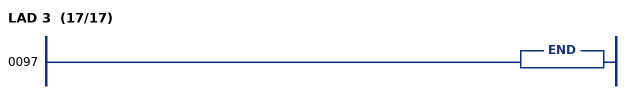
% Rung: 97 %
SOR END EOR

LADDER 4
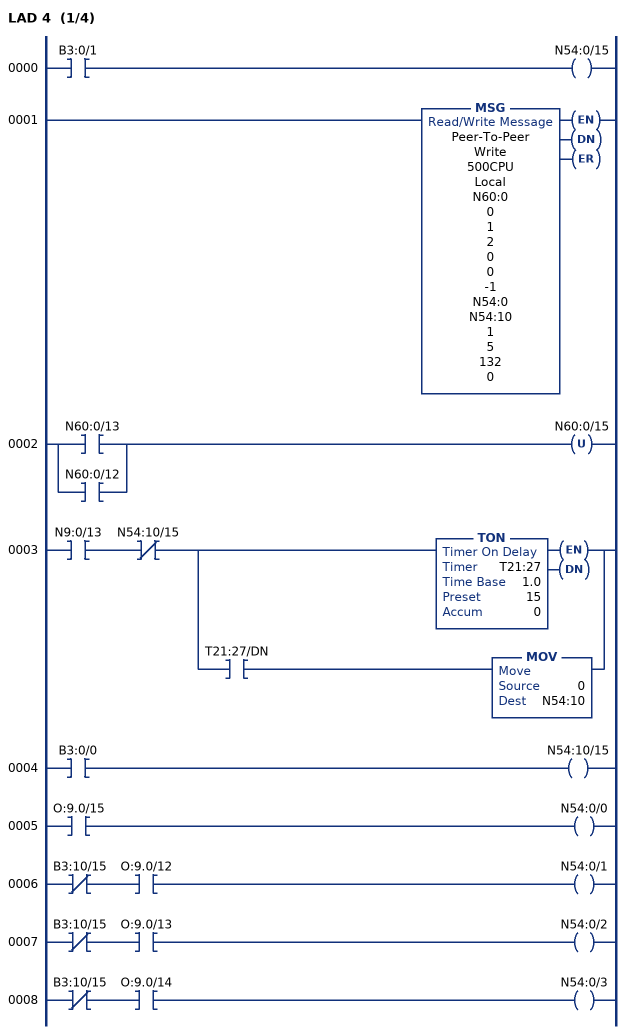
% Rung: 0 %
SOR XIC B3:0/1 OTE N54:0/15 EOR
% Rung: 1 %
SOR MSG Peer-To-Peer Write 500CPU Local N60:0 0 1 2 0 0 -1 N54:0 N54:10 1 5 132 0 EOR
%   MSG set-up: 500CPU Write | 5 | 1 | N54:10 | N54:0 | 0 | 2 | 2 | CLIENT | 0 | 0 %
% Rung: 2 %
SOR BST XIC N60:0/13 NXB XIC N60:0/12 BND OTU N60:0/15 EOR
% Rung: 3 %
SOR XIC N9:0/13 XIO N54:10/15 BST TON T21:27 1.0 15 0 NXB XIC T21:27/DN MOV 0 N54:10 BND EOR
% Rung: 4 %
SOR XIC B3:0/0 OTE N54:10/15 EOR
% Rung: 5 %
SOR XIC O:9.0/15 OTE N54:0/0 EOR
% Rung: 6 %
SOR XIO B3:10/15 XIC O:9.0/12 OTE N54:0/1 EOR
% Rung: 7 %
SOR XIO B3:10/15 XIC O:9.0/13 OTE N54:0/2 EOR
% Rung: 8 %
SOR XIO B3:10/15 XIC O:9.0/14 OTE N54:0/3 EOR

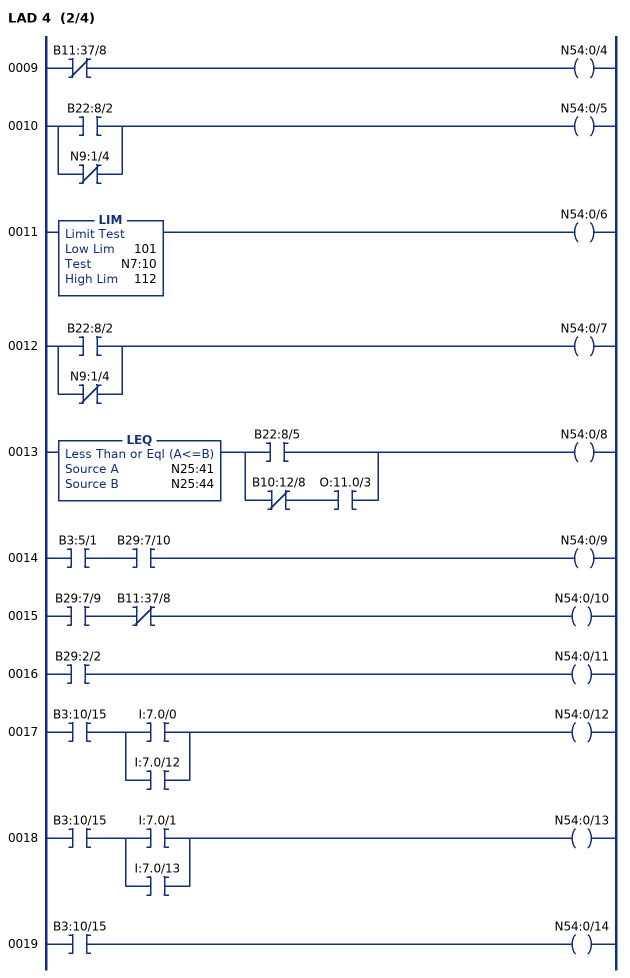
% Rung: 9 %
SOR XIO B11:37/8 OTE N54:0/4 EOR
% Rung: 10 %
SOR BST XIC B22:8/2 NXB XIO N9:1/4 BND OTE N54:0/5 EOR
% Rung: 11 %
SOR LIM 101 N7:10 112 OTE N54:0/6 EOR
% Rung: 12 %
SOR BST XIC B22:8/2 NXB XIO N9:1/4 BND OTE N54:0/7 EOR
% Rung: 13 %
SOR LEQ N25:41 N25:44 BST XIC B22:8/5 NXB XIO B10:12/8 XIC O:11.0/3 BND OTE N54:0/8 EOR
% Rung: 14 %
SOR XIC B3:5/1 XIC B29:7/10 OTE N54:0/9 EOR
% Rung: 15 %
SOR XIC B29:7/9 XIO B11:37/8 OTE N54:0/10 EOR
% Rung: 16 %
SOR XIC B29:2/2 OTE N54:0/11 EOR
% Rung: 17 %
SOR XIC B3:10/15 BST XIC I:7.0/0 NXB XIC I:7.0/12 BND OTE N54:0/12 EOR
% Rung: 18 %
SOR XIC B3:10/15 BST XIC I:7.0/1 NXB XIC I:7.0/13 BND OTE N54:0/13 EOR
% Rung: 19 %
SOR XIC B3:10/15 OTE N54:0/14 EOR

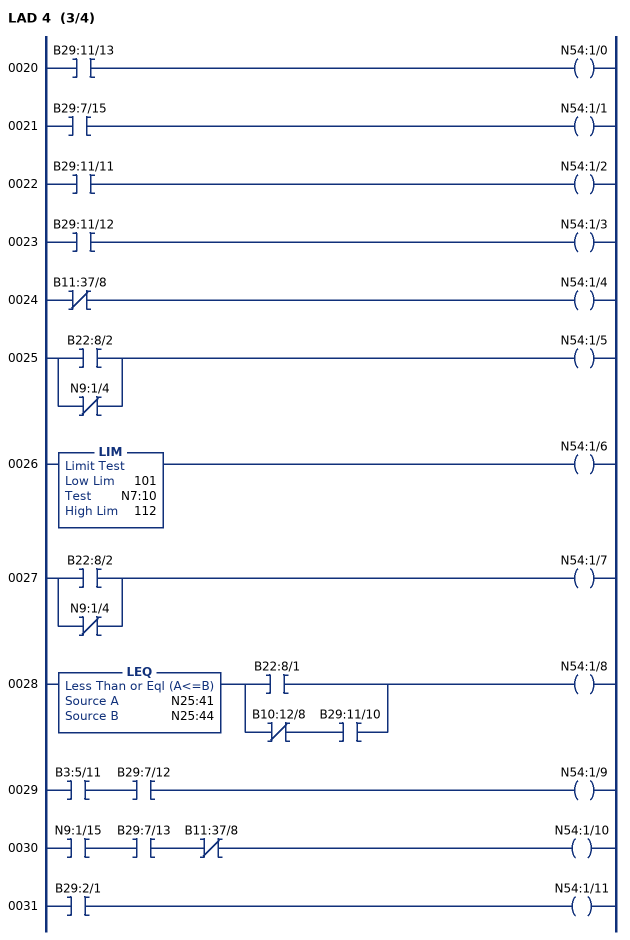
% Rung: 20 %
SOR XIC B29:11/13 OTE N54:1/0 EOR
% Rung: 21 %
SOR XIC B29:7/15 OTE N54:1/1 EOR
% Rung: 22 %
SOR XIC B29:11/11 OTE N54:1/2 EOR
% Rung: 23 %
SOR XIC B29:11/12 OTE N54:1/3 EOR
% Rung: 24 %
SOR XIO B11:37/8 OTE N54:1/4 EOR
% Rung: 25 %
SOR BST XIC B22:8/2 NXB XIO N9:1/4 BND OTE N54:1/5 EOR
% Rung: 26 %
SOR LIM 101 N7:10 112 OTE N54:1/6 EOR
% Rung: 27 %
SOR BST XIC B22:8/2 NXB XIO N9:1/4 BND OTE N54:1/7 EOR
% Rung: 28 %
SOR LEQ N25:41 N25:44 BST XIC B22:8/1 NXB XIO B10:12/8 XIC B29:11/10 BND OTE N54:1/8 EOR
% Rung: 29 %
SOR XIC B3:5/11 XIC B29:7/12 OTE N54:1/9 EOR
% Rung: 30 %
SOR XIC N9:1/15 XIC B29:7/13 XIO B11:37/8 OTE N54:1/10 EOR
% Rung: 31 %
SOR XIC B29:2/1 OTE N54:1/11 EOR

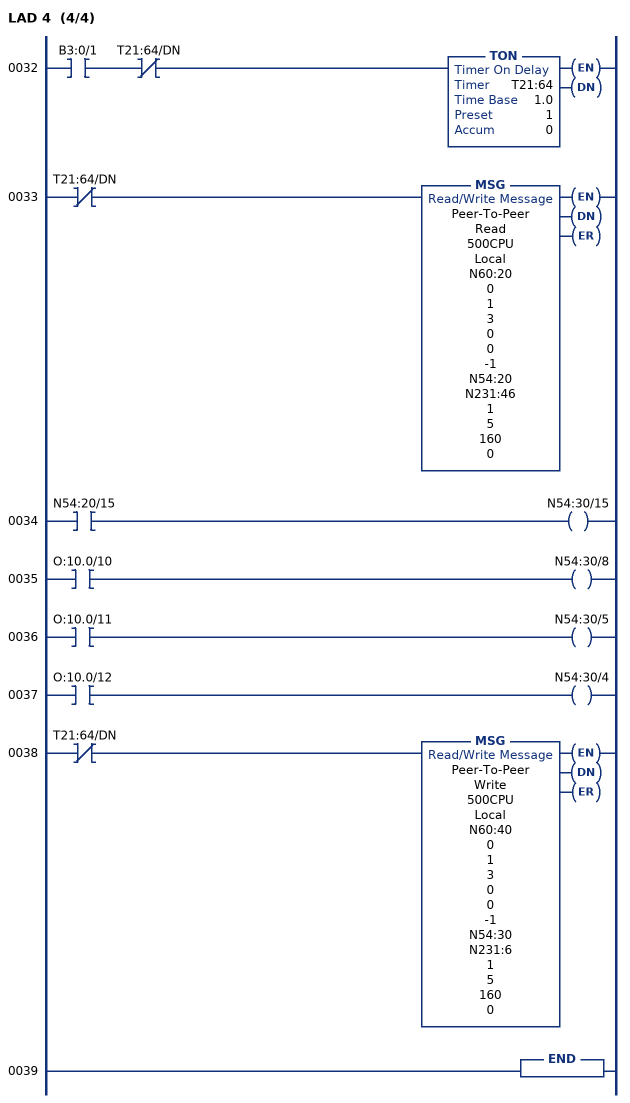
% Rung: 32 %
SOR XIC B3:0/1 XIO T21:64/DN TON T21:64 1.0 1 0 EOR
% Rung: 33 %
SOR XIO T21:64/DN MSG Peer-To-Peer Read 500CPU Local N60:20 0 1 3 0 0 -1 N54:20 N231:46 1 5 160 0 EOR
%   MSG set-up: 500CPU Read | 5 | 1 | N231:46 | N54:20 | 0 | 3 | 3 | CLIENT | 0 | 0 %
% Rung: 34 %
SOR XIC N54:20/15 OTE N54:30/15 EOR
% Rung: 35 %
SOR XIC O:10.0/10 OTE N54:30/8 EOR
% Rung: 36 %
SOR XIC O:10.0/11 OTE N54:30/5 EOR
% Rung: 37 %
SOR XIC O:10.0/12 OTE N54:30/4 EOR
% Rung: 38 %
SOR XIO T21:64/DN MSG Peer-To-Peer Write 500CPU Local N60:40 0 1 3 0 0 -1 N54:30 N231:6 1 5 160 0 EOR
%   MSG set-up: 500CPU Write | 5 | 1 | N231:6 | N54:30 | 0 | 3 | 3 | CLIENT | 0 | 0 %
% Rung: 39 %
SOR END EOR

LADDER 5
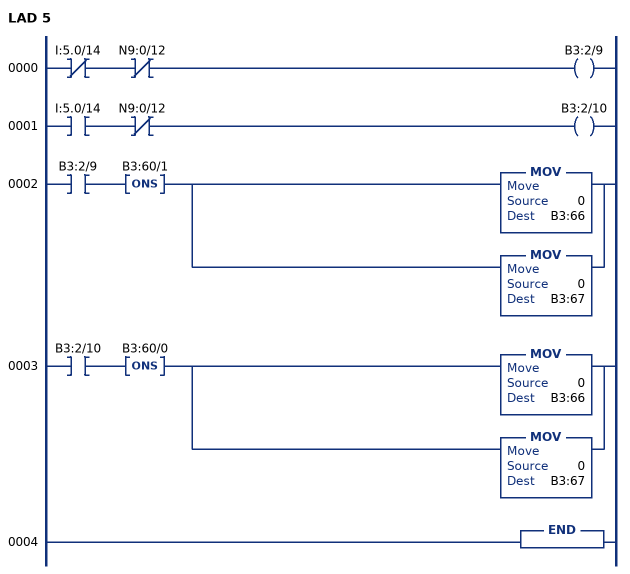
% Rung: 0 %
SOR XIO I:5.0/14 XIO N9:0/12 OTE B3:2/9 EOR
% Rung: 1 %
SOR XIC I:5.0/14 XIO N9:0/12 OTE B3:2/10 EOR
% Rung: 2 %
SOR XIC B3:2/9 OSR B3:60/1 BST MOV 0 B3:66 NXB MOV 0 B3:67 BND EOR
% Rung: 3 %
SOR XIC B3:2/10 OSR B3:60/0 BST MOV 0 B3:66 NXB MOV 0 B3:67 BND EOR
% Rung: 4 %
SOR END EOR

LADDER 6
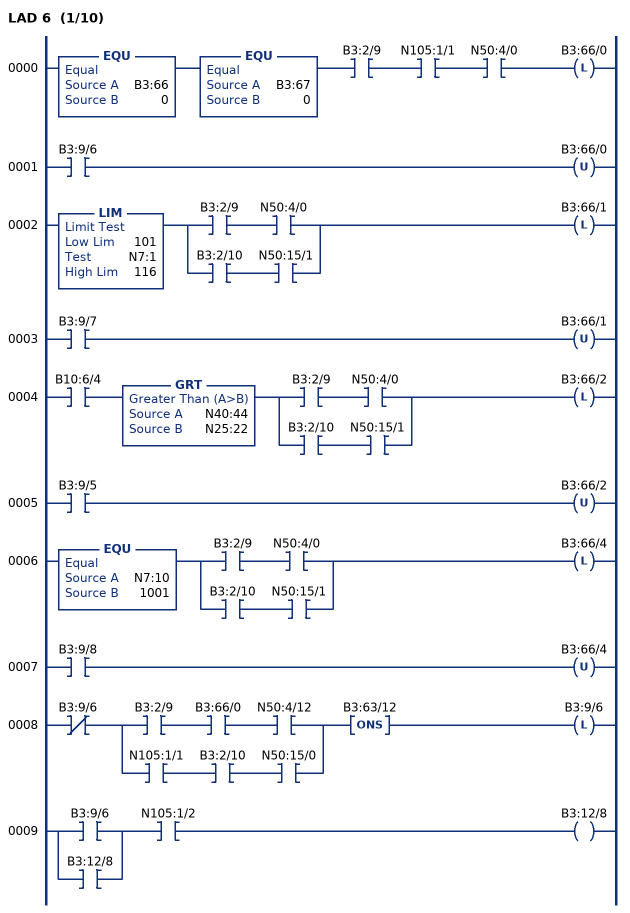
% Rung: 0 %
SOR EQU B3:66 0 EQU B3:67 0 XIC B3:2/9 XIC N105:1/1 XIC N50:4/0 OTL B3:66/0 EOR
% Rung: 1 %
SOR XIC B3:9/6 OTU B3:66/0 EOR
% Rung: 2 %
SOR LIM 101 N7:1 116 BST XIC B3:2/9 XIC N50:4/0 NXB XIC B3:2/10 XIC N50:15/1 BND OTL B3:66/1 EOR
% Rung: 3 %
SOR XIC B3:9/7 OTU B3:66/1 EOR
% Rung: 4 %
SOR XIC B10:6/4 GRT N40:44 N25:22 BST XIC B3:2/9 XIC N50:4/0 NXB XIC B3:2/10 XIC N50:15/1 BND OTL B3:66/2 EOR
% Rung: 5 %
SOR XIC B3:9/5 OTU B3:66/2 EOR
% Rung: 6 %
SOR EQU N7:10 1001 BST XIC B3:2/9 XIC N50:4/0 NXB XIC B3:2/10 XIC N50:15/1 BND OTL B3:66/4 EOR
% Rung: 7 %
SOR XIC B3:9/8 OTU B3:66/4 EOR
% Rung: 8 %
SOR XIO B3:9/6 BST XIC B3:2/9 XIC B3:66/0 XIC N50:4/12 NXB XIC N105:1/1 XIC B3:2/10 XIC N50:15/0 BND OSR B3:63/12 OTL B3:9/6 EOR
% Rung: 9 %
SOR BST XIC B3:9/6 NXB XIC B3:12/8 BND XIC N105:1/2 OTE B3:12/8 EOR

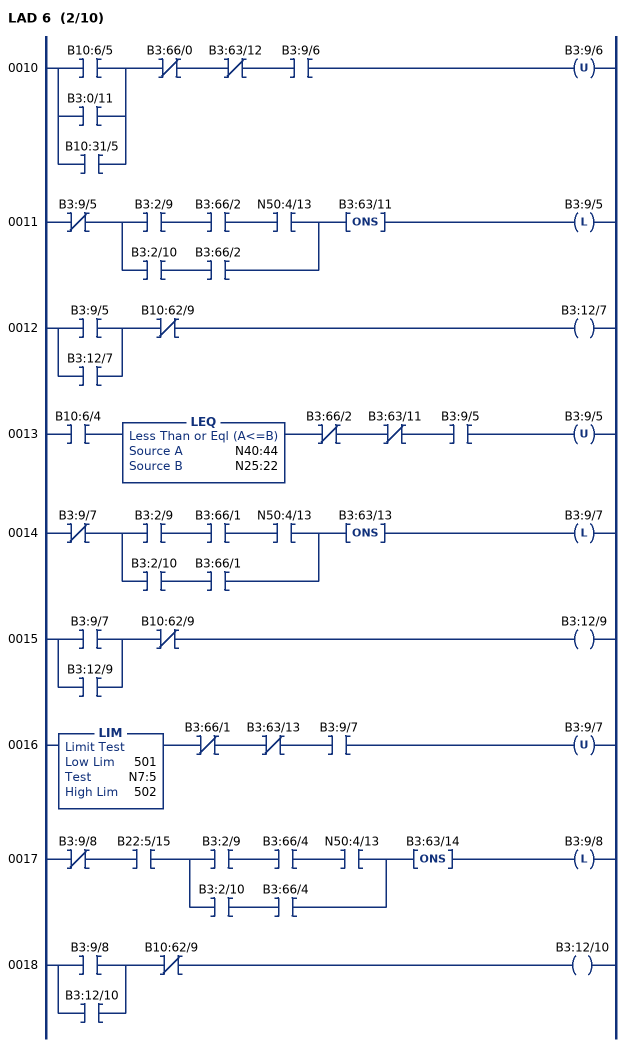
% Rung: 10 %
SOR BST XIC B10:6/5 NXB XIC B3:0/11 NXB XIC B10:31/5 BND XIO B3:66/0 XIO B3:63/12 XIC B3:9/6 OTU B3:9/6 EOR
% Rung: 11 %
SOR XIO B3:9/5 BST XIC B3:2/9 XIC B3:66/2 XIC N50:4/13 NXB XIC B3:2/10 XIC B3:66/2 BND OSR B3:63/11 OTL B3:9/5 EOR
% Rung: 12 %
SOR BST XIC B3:9/5 NXB XIC B3:12/7 BND XIO B10:62/9 OTE B3:12/7 EOR
% Rung: 13 %
SOR XIC B10:6/4 LEQ N40:44 N25:22 XIO B3:66/2 XIO B3:63/11 XIC B3:9/5 OTU B3:9/5 EOR
% Rung: 14 %
SOR XIO B3:9/7 BST XIC B3:2/9 XIC B3:66/1 XIC N50:4/13 NXB XIC B3:2/10 XIC B3:66/1 BND OSR B3:63/13 OTL B3:9/7 EOR
% Rung: 15 %
SOR BST XIC B3:9/7 NXB XIC B3:12/9 BND XIO B10:62/9 OTE B3:12/9 EOR
% Rung: 16 %
SOR LIM 501 N7:5 502 XIO B3:66/1 XIO B3:63/13 XIC B3:9/7 OTU B3:9/7 EOR
% Rung: 17 %
SOR XIO B3:9/8 XIC B22:5/15 BST XIC B3:2/9 XIC B3:66/4 XIC N50:4/13 NXB XIC B3:2/10 XIC B3:66/4 BND OSR B3:63/14 OTL B3:9/8 EOR
% Rung: 18 %
SOR BST XIC B3:9/8 NXB XIC B3:12/10 BND XIO B10:62/9 OTE B3:12/10 EOR

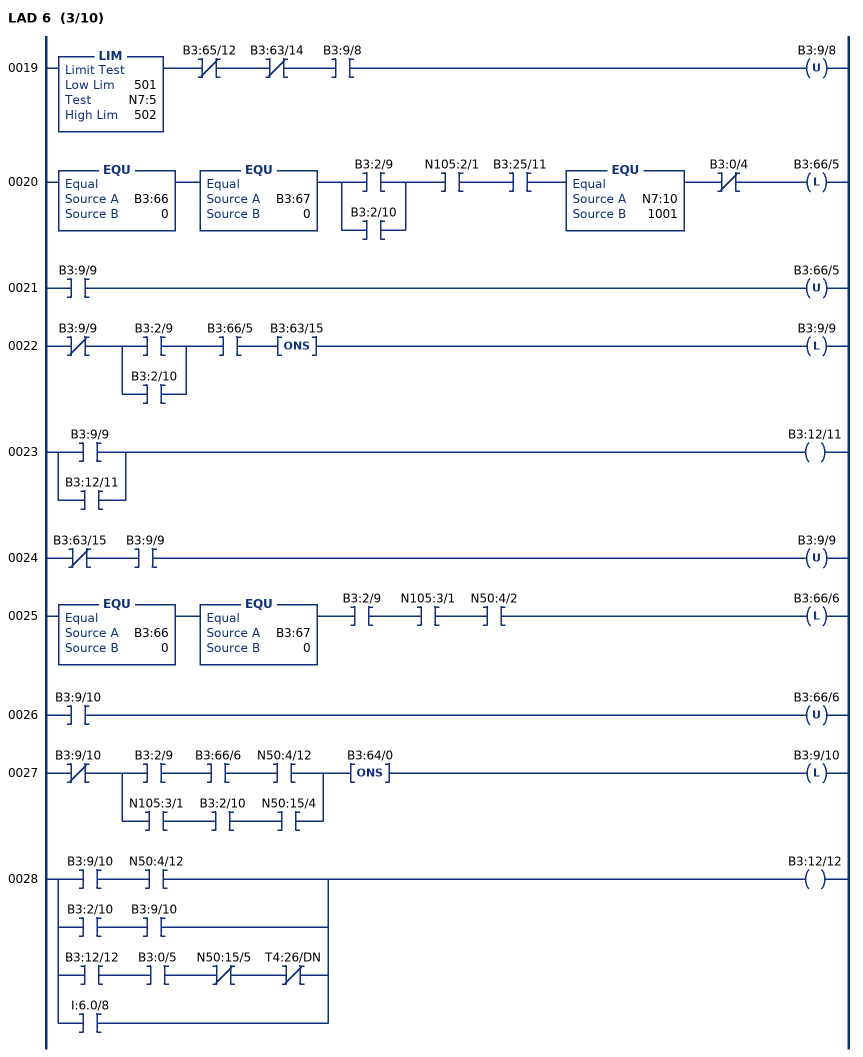
% Rung: 19 %
SOR LIM 501 N7:5 502 XIO B3:65/12 XIO B3:63/14 XIC B3:9/8 OTU B3:9/8 EOR
% Rung: 20 %
SOR EQU B3:66 0 EQU B3:67 0 BST XIC B3:2/9 NXB XIC B3:2/10 BND XIC N105:2/1 XIC B3:25/11 EQU N7:10 1001 XIO B3:0/4 OTL B3:66/5 EOR
% Rung: 21 %
SOR XIC B3:9/9 OTU B3:66/5 EOR
% Rung: 22 %
SOR XIO B3:9/9 BST XIC B3:2/9 NXB XIC B3:2/10 BND XIC B3:66/5 OSR B3:63/15 OTL B3:9/9 EOR
% Rung: 23 %
SOR BST XIC B3:9/9 NXB XIC B3:12/11 BND OTE B3:12/11 EOR
% Rung: 24 %
SOR XIO B3:63/15 XIC B3:9/9 OTU B3:9/9 EOR
% Rung: 25 %
SOR EQU B3:66 0 EQU B3:67 0 XIC B3:2/9 XIC N105:3/1 XIC N50:4/2 OTL B3:66/6 EOR
% Rung: 26 %
SOR XIC B3:9/10 OTU B3:66/6 EOR
% Rung: 27 %
SOR XIO B3:9/10 BST XIC B3:2/9 XIC B3:66/6 XIC N50:4/12 NXB XIC N105:3/1 XIC B3:2/10 XIC N50:15/4 BND OSR B3:64/0 OTL B3:9/10 EOR
% Rung: 28 %
SOR BST XIC B3:9/10 XIC N50:4/12 NXB XIC B3:2/10 XIC B3:9/10 NXB XIC B3:12/12 XIC B3:0/5 XIO N50:15/5 XIO T4:26/DN NXB XIC I:6.0/8 BND OTE B3:12/12 EOR

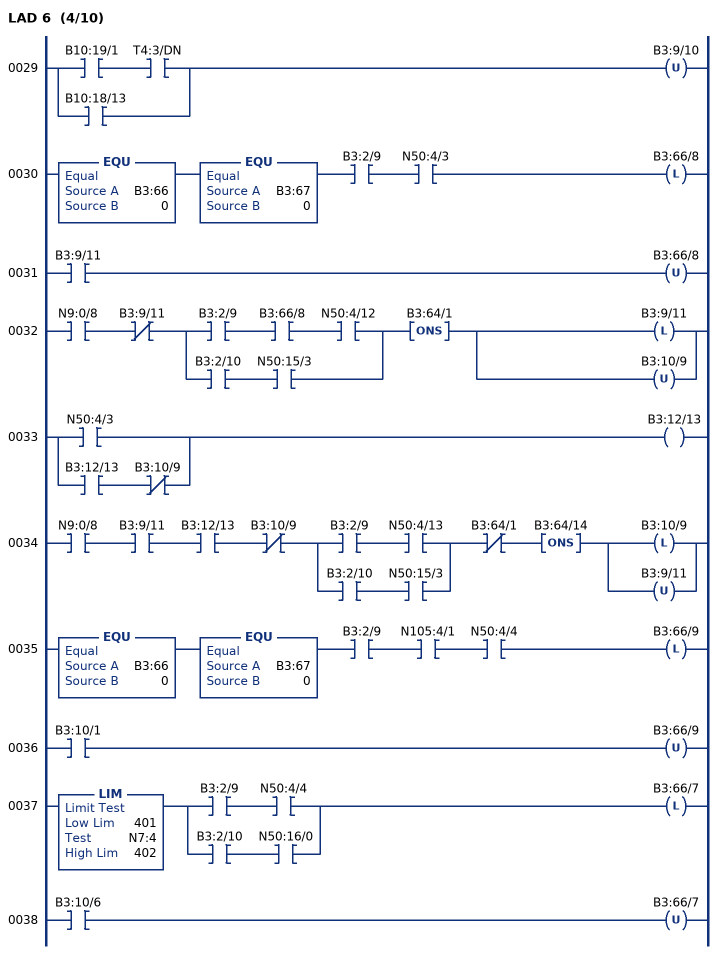
% Rung: 29 %
SOR BST XIC B10:19/1 XIC T4:3/DN NXB XIC B10:18/13 BND OTU B3:9/10 EOR
% Rung: 30 %
SOR EQU B3:66 0 EQU B3:67 0 XIC B3:2/9 XIC N50:4/3 OTL B3:66/8 EOR
% Rung: 31 %
SOR XIC B3:9/11 OTU B3:66/8 EOR
% Rung: 32 %
SOR XIC N9:0/8 XIO B3:9/11 BST XIC B3:2/9 XIC B3:66/8 XIC N50:4/12 NXB XIC B3:2/10 XIC N50:15/3 BND OSR B3:64/1 BST OTL B3:9/11 NXB OTU B3:10/9 BND EOR
% Rung: 33 %
SOR BST XIC N50:4/3 NXB XIC B3:12/13 XIO B3:10/9 BND OTE B3:12/13 EOR
% Rung: 34 %
SOR XIC N9:0/8 XIC B3:9/11 XIC B3:12/13 XIO B3:10/9 BST XIC B3:2/9 XIC N50:4/13 NXB XIC B3:2/10 XIC N50:15/3 BND XIO B3:64/1 OSR B3:64/14 BST OTL B3:10/9 NXB OTU B3:9/11 BND EOR
% Rung: 35 %
SOR EQU B3:66 0 EQU B3:67 0 XIC B3:2/9 XIC N105:4/1 XIC N50:4/4 OTL B3:66/9 EOR
% Rung: 36 %
SOR XIC B3:10/1 OTU B3:66/9 EOR
% Rung: 37 %
SOR LIM 401 N7:4 402 BST XIC B3:2/9 XIC N50:4/4 NXB XIC B3:2/10 XIC N50:16/0 BND OTL B3:66/7 EOR
% Rung: 38 %
SOR XIC B3:10/6 OTU B3:66/7 EOR

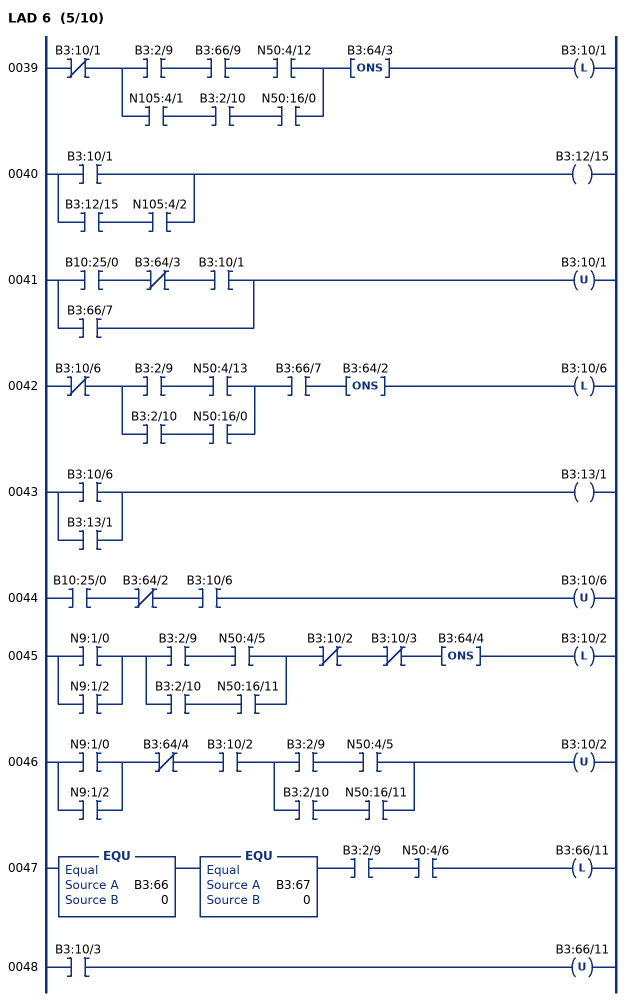
% Rung: 39 %
SOR XIO B3:10/1 BST XIC B3:2/9 XIC B3:66/9 XIC N50:4/12 NXB XIC N105:4/1 XIC B3:2/10 XIC N50:16/0 BND OSR B3:64/3 OTL B3:10/1 EOR
% Rung: 40 %
SOR BST XIC B3:10/1 NXB XIC B3:12/15 XIC N105:4/2 BND OTE B3:12/15 EOR
% Rung: 41 %
SOR BST XIC B10:25/0 XIO B3:64/3 XIC B3:10/1 NXB XIC B3:66/7 BND OTU B3:10/1 EOR
% Rung: 42 %
SOR XIO B3:10/6 BST XIC B3:2/9 XIC N50:4/13 NXB XIC B3:2/10 XIC N50:16/0 BND XIC B3:66/7 OSR B3:64/2 OTL B3:10/6 EOR
% Rung: 43 %
SOR BST XIC B3:10/6 NXB XIC B3:13/1 BND OTE B3:13/1 EOR
% Rung: 44 %
SOR XIC B10:25/0 XIO B3:64/2 XIC B3:10/6 OTU B3:10/6 EOR
% Rung: 45 %
SOR BST XIC N9:1/0 NXB XIC N9:1/2 BND BST XIC B3:2/9 XIC N50:4/5 NXB XIC B3:2/10 XIC N50:16/11 BND XIO B3:10/2 XIO B3:10/3 OSR B3:64/4 OTL B3:10/2 EOR
% Rung: 46 %
SOR BST XIC N9:1/0 NXB XIC N9:1/2 BND XIO B3:64/4 XIC B3:10/2 BST XIC B3:2/9 XIC N50:4/5 NXB XIC B3:2/10 XIC N50:16/11 BND OTU B3:10/2 EOR
% Rung: 47 %
SOR EQU B3:66 0 EQU B3:67 0 XIC B3:2/9 XIC N50:4/6 OTL B3:66/11 EOR
% Rung: 48 %
SOR XIC B3:10/3 OTU B3:66/11 EOR

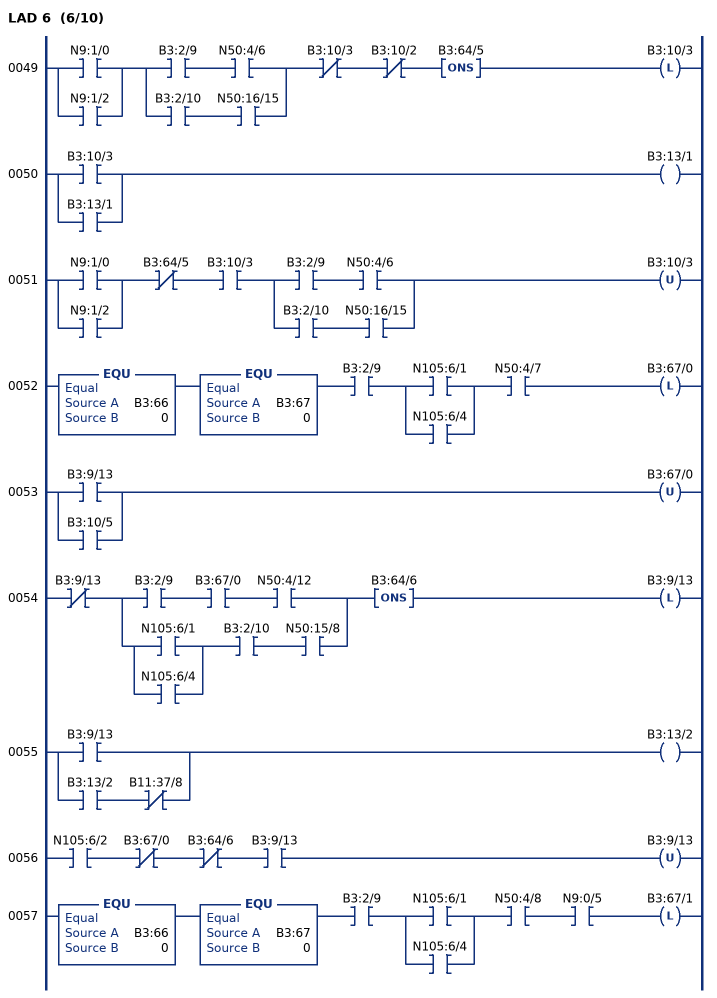
% Rung: 49 %
SOR BST XIC N9:1/0 NXB XIC N9:1/2 BND BST XIC B3:2/9 XIC N50:4/6 NXB XIC B3:2/10 XIC N50:16/15 BND XIO B3:10/3 XIO B3:10/2 OSR B3:64/5 OTL B3:10/3 EOR
% Rung: 50 %
SOR BST XIC B3:10/3 NXB XIC B3:13/1 BND OTE B3:13/1 EOR
% Rung: 51 %
SOR BST XIC N9:1/0 NXB XIC N9:1/2 BND XIO B3:64/5 XIC B3:10/3 BST XIC B3:2/9 XIC N50:4/6 NXB XIC B3:2/10 XIC N50:16/15 BND OTU B3:10/3 EOR
% Rung: 52 %
SOR EQU B3:66 0 EQU B3:67 0 XIC B3:2/9 BST XIC N105:6/1 NXB XIC N105:6/4 BND XIC N50:4/7 OTL B3:67/0 EOR
% Rung: 53 %
SOR BST XIC B3:9/13 NXB XIC B3:10/5 BND OTU B3:67/0 EOR
% Rung: 54 %
SOR XIO B3:9/13 BST XIC B3:2/9 XIC B3:67/0 XIC N50:4/12 NXB BST XIC N105:6/1 NXB XIC N105:6/4 BND XIC B3:2/10 XIC N50:15/8 BND OSR B3:64/6 OTL B3:9/13 EOR
% Rung: 55 %
SOR BST XIC B3:9/13 NXB XIC B3:13/2 XIO B11:37/8 BND OTE B3:13/2 EOR
% Rung: 56 %
SOR XIC N105:6/2 XIO B3:67/0 XIO B3:64/6 XIC B3:9/13 OTU B3:9/13 EOR
% Rung: 57 %
SOR EQU B3:66 0 EQU B3:67 0 XIC B3:2/9 BST XIC N105:6/1 NXB XIC N105:6/4 BND XIC N50:4/8 XIC N9:0/5 OTL B3:67/1 EOR

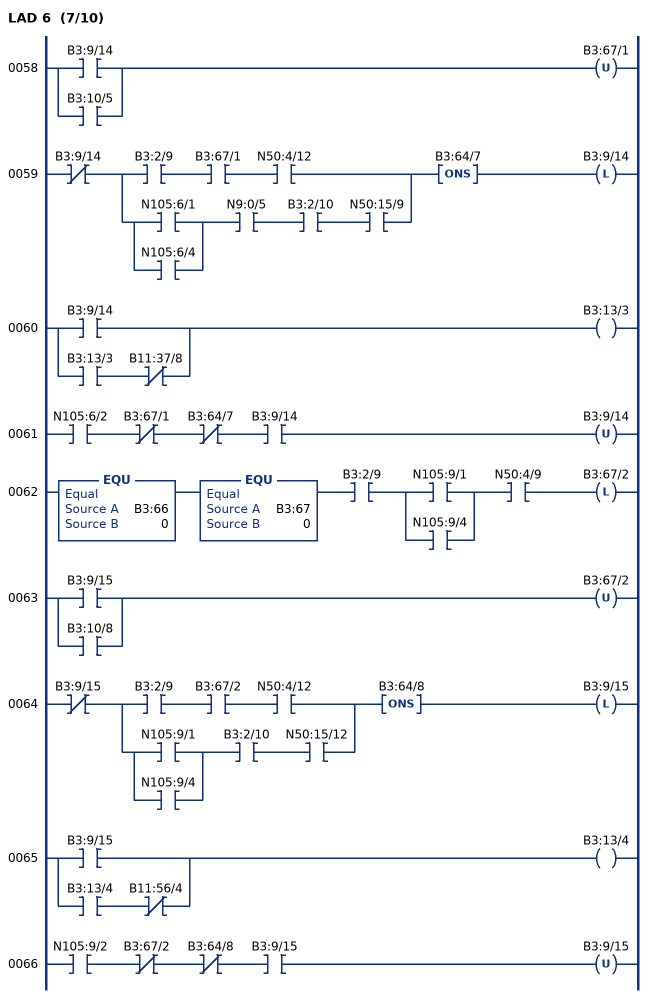
% Rung: 58 %
SOR BST XIC B3:9/14 NXB XIC B3:10/5 BND OTU B3:67/1 EOR
% Rung: 59 %
SOR XIO B3:9/14 BST XIC B3:2/9 XIC B3:67/1 XIC N50:4/12 NXB BST XIC N105:6/1 NXB XIC N105:6/4 BND XIC N9:0/5 XIC B3:2/10 XIC N50:15/9 BND OSR B3:64/7 OTL B3:9/14 EOR
% Rung: 60 %
SOR BST XIC B3:9/14 NXB XIC B3:13/3 XIO B11:37/8 BND OTE B3:13/3 EOR
% Rung: 61 %
SOR XIC N105:6/2 XIO B3:67/1 XIO B3:64/7 XIC B3:9/14 OTU B3:9/14 EOR
% Rung: 62 %
SOR EQU B3:66 0 EQU B3:67 0 XIC B3:2/9 BST XIC N105:9/1 NXB XIC N105:9/4 BND XIC N50:4/9 OTL B3:67/2 EOR
% Rung: 63 %
SOR BST XIC B3:9/15 NXB XIC B3:10/8 BND OTU B3:67/2 EOR
% Rung: 64 %
SOR XIO B3:9/15 BST XIC B3:2/9 XIC B3:67/2 XIC N50:4/12 NXB BST XIC N105:9/1 NXB XIC N105:9/4 BND XIC B3:2/10 XIC N50:15/12 BND OSR B3:64/8 OTL B3:9/15 EOR
% Rung: 65 %
SOR BST XIC B3:9/15 NXB XIC B3:13/4 XIO B11:56/4 BND OTE B3:13/4 EOR
% Rung: 66 %
SOR XIC N105:9/2 XIO B3:67/2 XIO B3:64/8 XIC B3:9/15 OTU B3:9/15 EOR

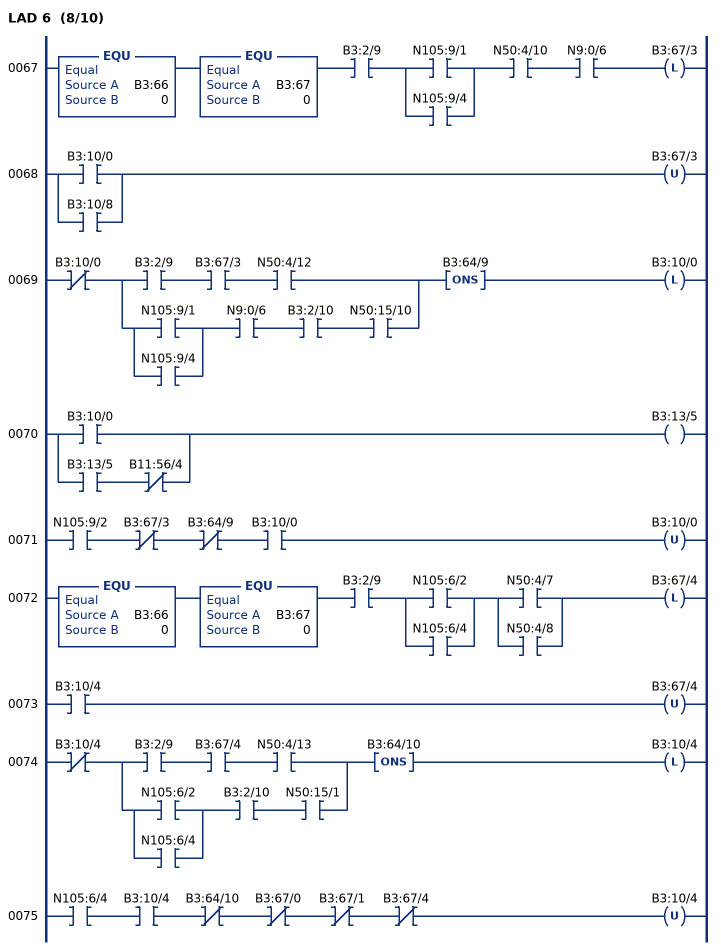
% Rung: 67 %
SOR EQU B3:66 0 EQU B3:67 0 XIC B3:2/9 BST XIC N105:9/1 NXB XIC N105:9/4 BND XIC N50:4/10 XIC N9:0/6 OTL B3:67/3 EOR
% Rung: 68 %
SOR BST XIC B3:10/0 NXB XIC B3:10/8 BND OTU B3:67/3 EOR
% Rung: 69 %
SOR XIO B3:10/0 BST XIC B3:2/9 XIC B3:67/3 XIC N50:4/12 NXB BST XIC N105:9/1 NXB XIC N105:9/4 BND XIC N9:0/6 XIC B3:2/10 XIC N50:15/10 BND OSR B3:64/9 OTL B3:10/0 EOR
% Rung: 70 %
SOR BST XIC B3:10/0 NXB XIC B3:13/5 XIO B11:56/4 BND OTE B3:13/5 EOR
% Rung: 71 %
SOR XIC N105:9/2 XIO B3:67/3 XIO B3:64/9 XIC B3:10/0 OTU B3:10/0 EOR
% Rung: 72 %
SOR EQU B3:66 0 EQU B3:67 0 XIC B3:2/9 BST XIC N105:6/2 NXB XIC N105:6/4 BND BST XIC N50:4/7 NXB XIC N50:4/8 BND OTL B3:67/4 EOR
% Rung: 73 %
SOR XIC B3:10/4 OTU B3:67/4 EOR
% Rung: 74 %
SOR XIO B3:10/4 BST XIC B3:2/9 XIC B3:67/4 XIC N50:4/13 NXB BST XIC N105:6/2 NXB XIC N105:6/4 BND XIC B3:2/10 XIC N50:15/1 BND OSR B3:64/10 OTL B3:10/4 EOR
% Rung: 75 %
SOR XIC N105:6/4 XIC B3:10/4 XIO B3:64/10 XIO B3:67/0 XIO B3:67/1 XIO B3:67/4 OTU B3:10/4 EOR

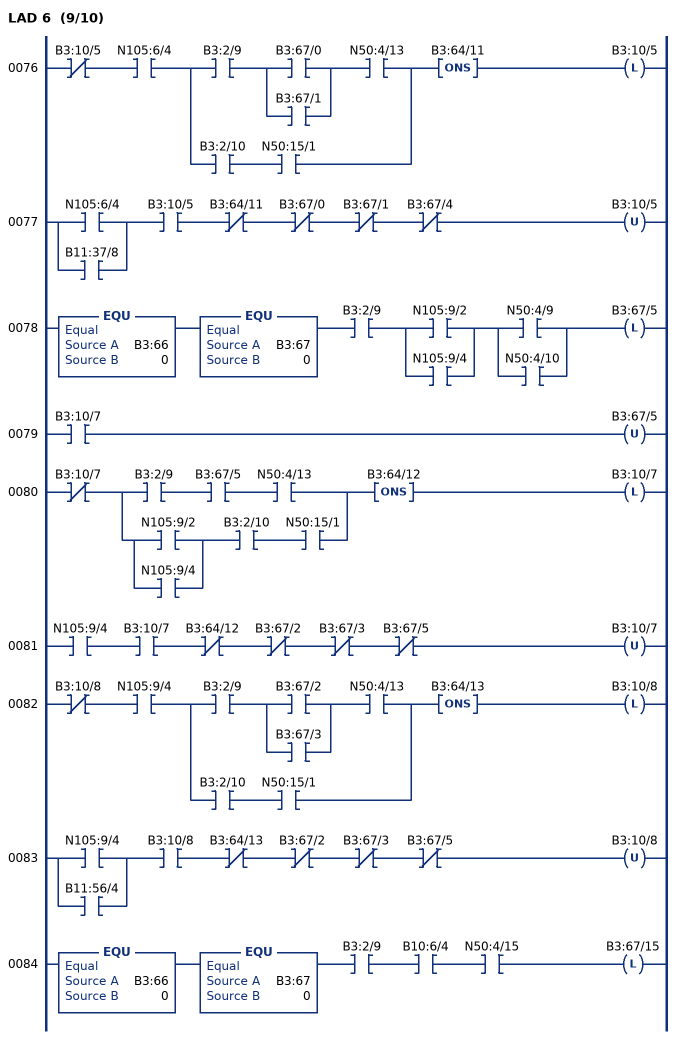
% Rung: 76 %
SOR XIO B3:10/5 XIC N105:6/4 BST XIC B3:2/9 BST XIC B3:67/0 NXB XIC B3:67/1 BND XIC N50:4/13 NXB XIC B3:2/10 XIC N50:15/1 BND OSR B3:64/11 OTL B3:10/5 EOR
% Rung: 77 %
SOR BST XIC N105:6/4 NXB XIC B11:37/8 BND XIC B3:10/5 XIO B3:64/11 XIO B3:67/0 XIO B3:67/1 XIO B3:67/4 OTU B3:10/5 EOR
% Rung: 78 %
SOR EQU B3:66 0 EQU B3:67 0 XIC B3:2/9 BST XIC N105:9/2 NXB XIC N105:9/4 BND BST XIC N50:4/9 NXB XIC N50:4/10 BND OTL B3:67/5 EOR
% Rung: 79 %
SOR XIC B3:10/7 OTU B3:67/5 EOR
% Rung: 80 %
SOR XIO B3:10/7 BST XIC B3:2/9 XIC B3:67/5 XIC N50:4/13 NXB BST XIC N105:9/2 NXB XIC N105:9/4 BND XIC B3:2/10 XIC N50:15/1 BND OSR B3:64/12 OTL B3:10/7 EOR
% Rung: 81 %
SOR XIC N105:9/4 XIC B3:10/7 XIO B3:64/12 XIO B3:67/2 XIO B3:67/3 XIO B3:67/5 OTU B3:10/7 EOR
% Rung: 82 %
SOR XIO B3:10/8 XIC N105:9/4 BST XIC B3:2/9 BST XIC B3:67/2 NXB XIC B3:67/3 BND XIC N50:4/13 NXB XIC B3:2/10 XIC N50:15/1 BND OSR B3:64/13 OTL B3:10/8 EOR
% Rung: 83 %
SOR BST XIC N105:9/4 NXB XIC B11:56/4 BND XIC B3:10/8 XIO B3:64/13 XIO B3:67/2 XIO B3:67/3 XIO B3:67/5 OTU B3:10/8 EOR
% Rung: 84 %
SOR EQU B3:66 0 EQU B3:67 0 XIC B3:2/9 XIC B10:6/4 XIC N50:4/15 OTL B3:67/15 EOR

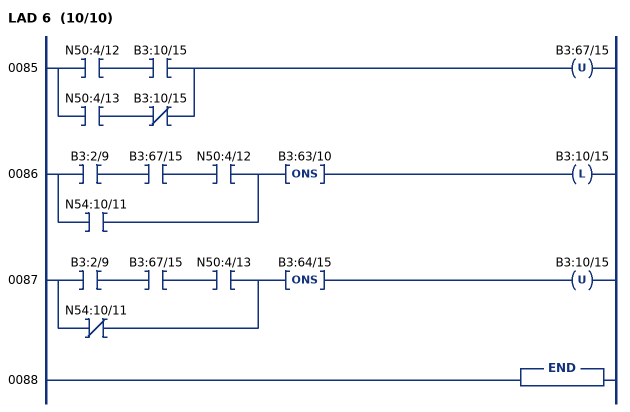
% Rung: 85 %
SOR BST XIC N50:4/12 XIC B3:10/15 NXB XIC N50:4/13 XIO B3:10/15 BND OTU B3:67/15 EOR
% Rung: 86 %
SOR BST XIC B3:2/9 XIC B3:67/15 XIC N50:4/12 NXB XIC N54:10/11 BND OSR B3:63/10 OTL B3:10/15 EOR
% Rung: 87 %
SOR BST XIC B3:2/9 XIC B3:67/15 XIC N50:4/13 NXB XIO N54:10/11 BND OSR B3:64/15 OTU B3:10/15 EOR
% Rung: 88 %
SOR END EOR

LADDER 9
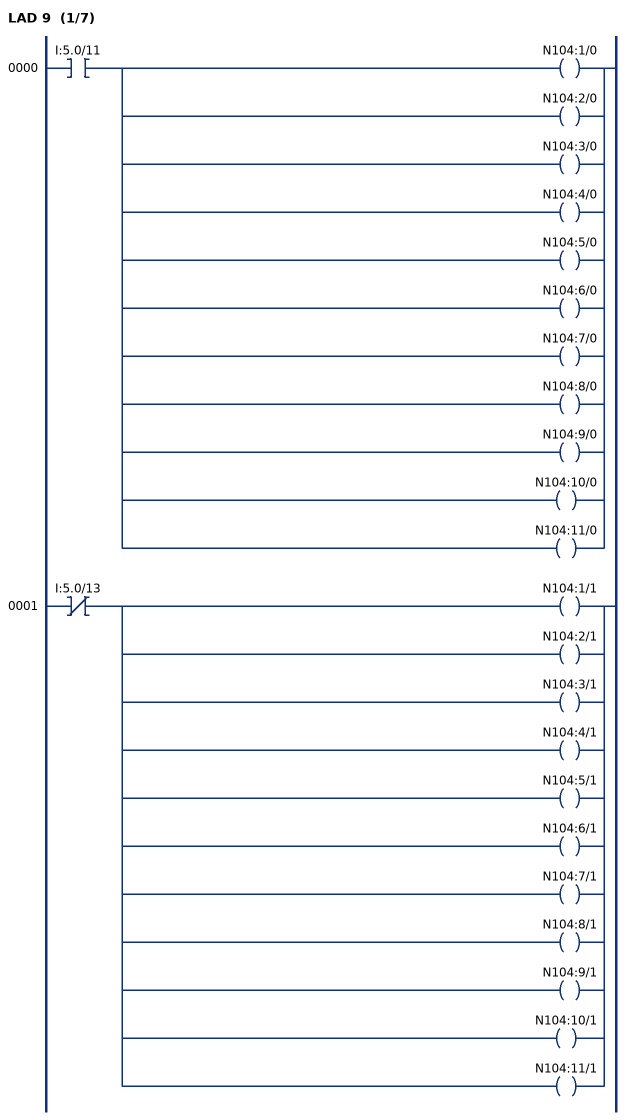
% Rung: 0 %
SOR XIC I:5.0/11 BST OTE N104:1/0 NXB OTE N104:2/0 NXB OTE N104:3/0 NXB OTE N104:4/0 NXB OTE N104:5/0 NXB OTE N104:6/0 NXB OTE N104:7/0 NXB OTE N104:8/0 NXB OTE N104:9/0 NXB OTE N104:10/0 NXB OTE N104:11/0 BND EOR
% Rung: 1 %
SOR XIO I:5.0/13 BST OTE N104:1/1 NXB OTE N104:2/1 NXB OTE N104:3/1 NXB OTE N104:4/1 NXB OTE N104:5/1 NXB OTE N104:6/1 NXB OTE N104:7/1 NXB OTE N104:8/1 NXB OTE N104:9/1 NXB OTE N104:10/1 NXB OTE N104:11/1 BND EOR

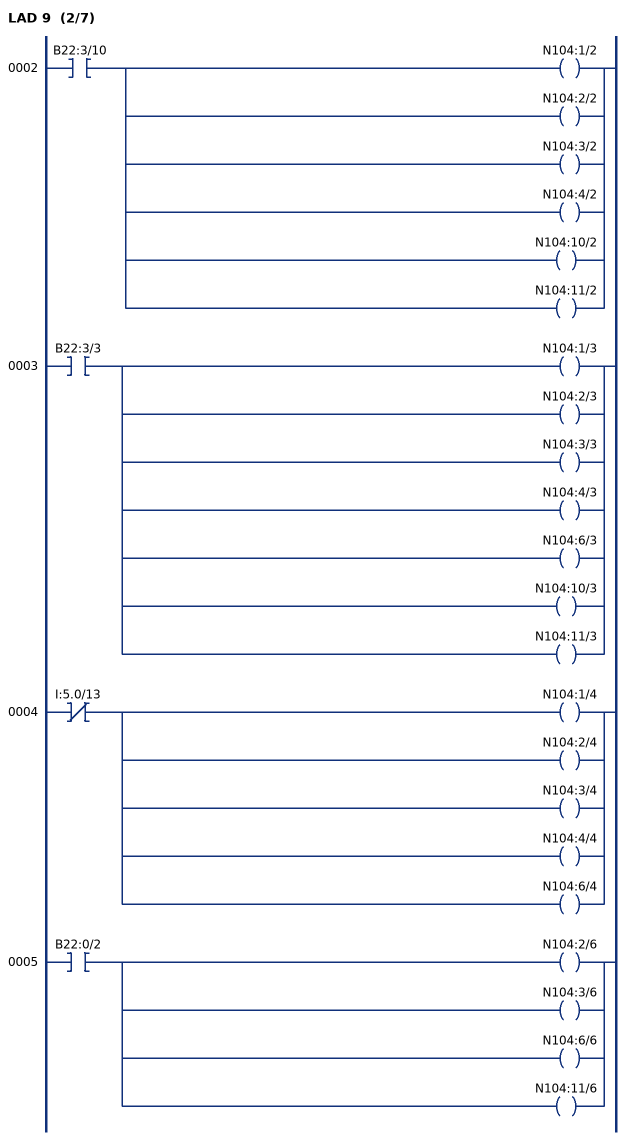
% Rung: 2 %
SOR XIC B22:3/10 BST OTE N104:1/2 NXB OTE N104:2/2 NXB OTE N104:3/2 NXB OTE N104:4/2 NXB OTE N104:10/2 NXB OTE N104:11/2 BND EOR
% Rung: 3 %
SOR XIC B22:3/3 BST OTE N104:1/3 NXB OTE N104:2/3 NXB OTE N104:3/3 NXB OTE N104:4/3 NXB OTE N104:6/3 NXB OTE N104:10/3 NXB OTE N104:11/3 BND EOR
% Rung: 4 %
SOR XIO I:5.0/13 BST OTE N104:1/4 NXB OTE N104:2/4 NXB OTE N104:3/4 NXB OTE N104:4/4 NXB OTE N104:6/4 BND EOR
% Rung: 5 %
SOR XIC B22:0/2 BST OTE N104:2/6 NXB OTE N104:3/6 NXB OTE N104:6/6 NXB OTE N104:11/6 BND EOR

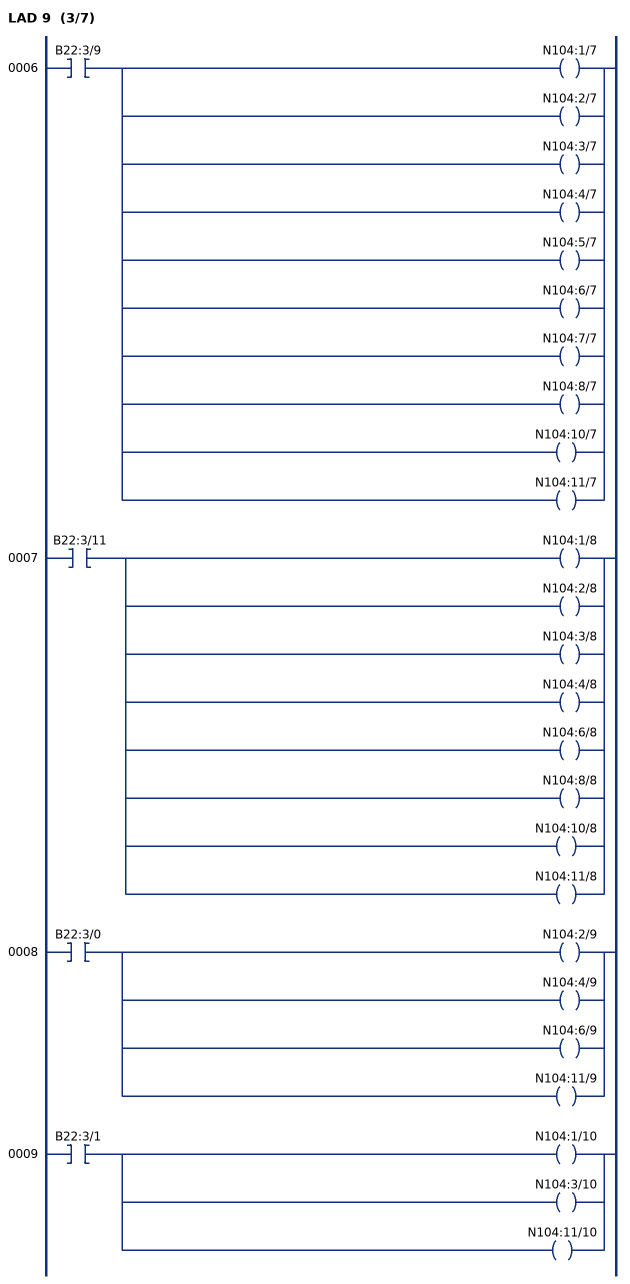
% Rung: 6 %
SOR XIC B22:3/9 BST OTE N104:1/7 NXB OTE N104:2/7 NXB OTE N104:3/7 NXB OTE N104:4/7 NXB OTE N104:5/7 NXB OTE N104:6/7 NXB OTE N104:7/7 NXB OTE N104:8/7 NXB OTE N104:10/7 NXB OTE N104:11/7 BND EOR
% Rung: 7 %
SOR XIC B22:3/11 BST OTE N104:1/8 NXB OTE N104:2/8 NXB OTE N104:3/8 NXB OTE N104:4/8 NXB OTE N104:6/8 NXB OTE N104:8/8 NXB OTE N104:10/8 NXB OTE N104:11/8 BND EOR
% Rung: 8 %
SOR XIC B22:3/0 BST OTE N104:2/9 NXB OTE N104:4/9 NXB OTE N104:6/9 NXB OTE N104:11/9 BND EOR
% Rung: 9 %
SOR XIC B22:3/1 BST OTE N104:1/10 NXB OTE N104:3/10 NXB OTE N104:11/10 BND EOR

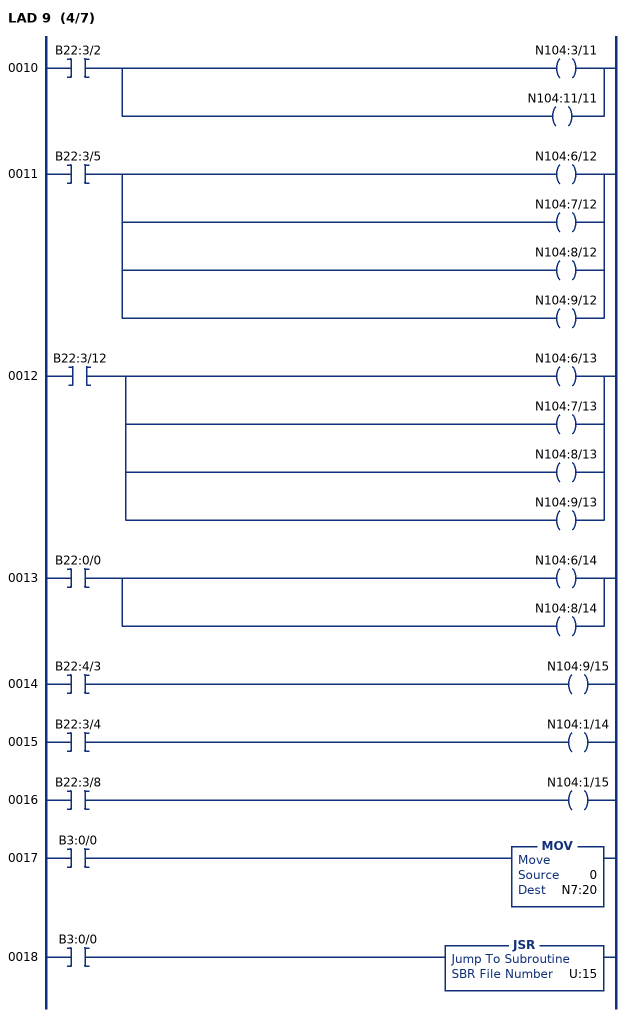
% Rung: 10 %
SOR XIC B22:3/2 BST OTE N104:3/11 NXB OTE N104:11/11 BND EOR
% Rung: 11 %
SOR XIC B22:3/5 BST OTE N104:6/12 NXB OTE N104:7/12 NXB OTE N104:8/12 NXB OTE N104:9/12 BND EOR
% Rung: 12 %
SOR XIC B22:3/12 BST OTE N104:6/13 NXB OTE N104:7/13 NXB OTE N104:8/13 NXB OTE N104:9/13 BND EOR
% Rung: 13 %
SOR XIC B22:0/0 BST OTE N104:6/14 NXB OTE N104:8/14 BND EOR
% Rung: 14 %
SOR XIC B22:4/3 OTE N104:9/15 EOR
% Rung: 15 %
SOR XIC B22:3/4 OTE N104:1/14 EOR
% Rung: 16 %
SOR XIC B22:3/8 OTE N104:1/15 EOR
% Rung: 17 %
SOR XIC B3:0/0 MOV 0 N7:20 EOR
% Rung: 18 %
SOR XIC B3:0/0 JSR U:15 EOR

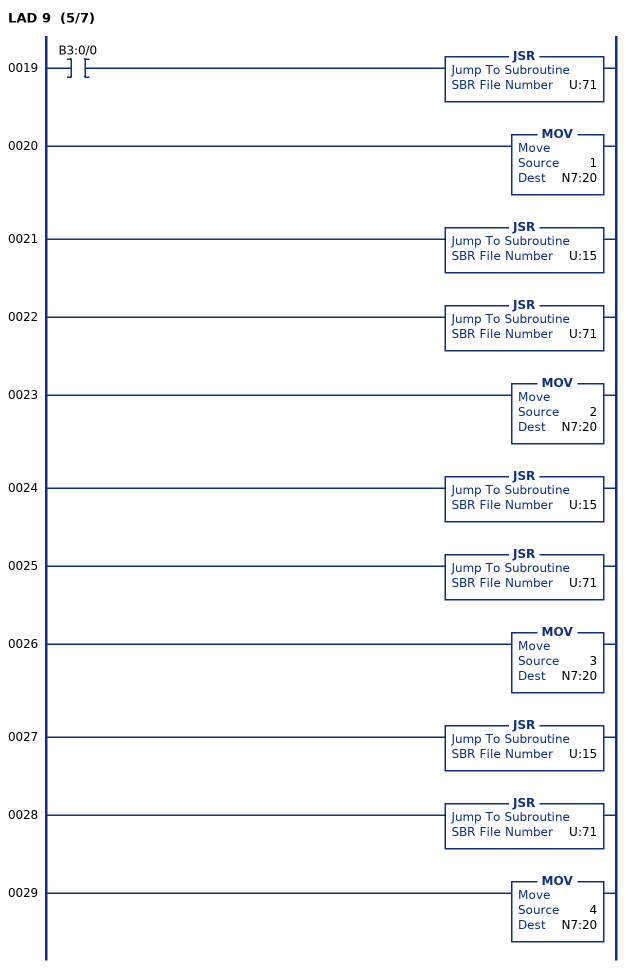
% Rung: 19 %
SOR XIC B3:0/0 JSR U:71 EOR
% Rung: 20 %
SOR MOV 1 N7:20 EOR
% Rung: 21 %
SOR JSR U:15 EOR
% Rung: 22 %
SOR JSR U:71 EOR
% Rung: 23 %
SOR MOV 2 N7:20 EOR
% Rung: 24 %
SOR JSR U:15 EOR
% Rung: 25 %
SOR JSR U:71 EOR
% Rung: 26 %
SOR MOV 3 N7:20 EOR
% Rung: 27 %
SOR JSR U:15 EOR
% Rung: 28 %
SOR JSR U:71 EOR
% Rung: 29 %
SOR MOV 4 N7:20 EOR

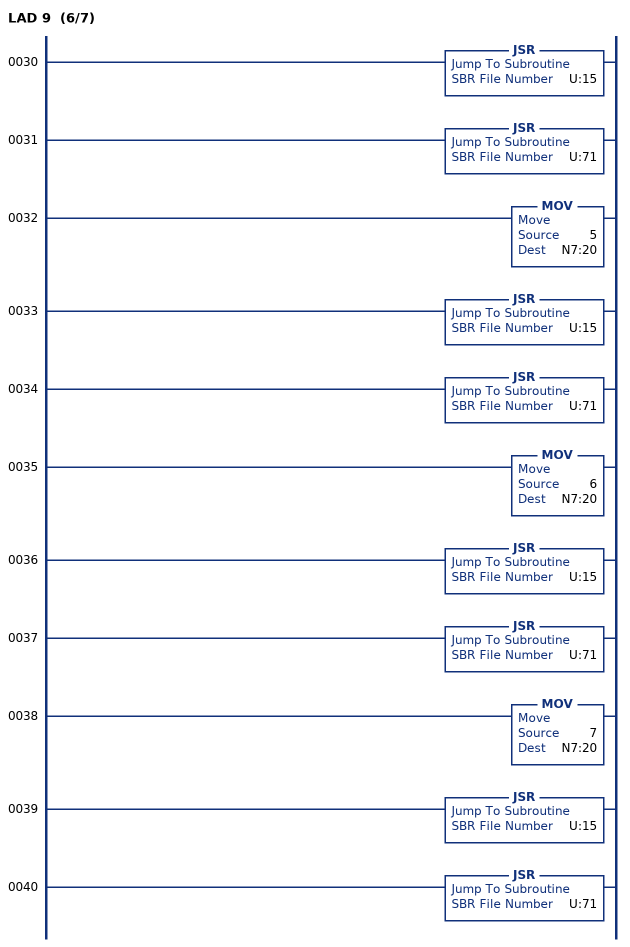
% Rung: 30 %
SOR JSR U:15 EOR
% Rung: 31 %
SOR JSR U:71 EOR
% Rung: 32 %
SOR MOV 5 N7:20 EOR
% Rung: 33 %
SOR JSR U:15 EOR
% Rung: 34 %
SOR JSR U:71 EOR
% Rung: 35 %
SOR MOV 6 N7:20 EOR
% Rung: 36 %
SOR JSR U:15 EOR
% Rung: 37 %
SOR JSR U:71 EOR
% Rung: 38 %
SOR MOV 7 N7:20 EOR
% Rung: 39 %
SOR JSR U:15 EOR
% Rung: 40 %
SOR JSR U:71 EOR

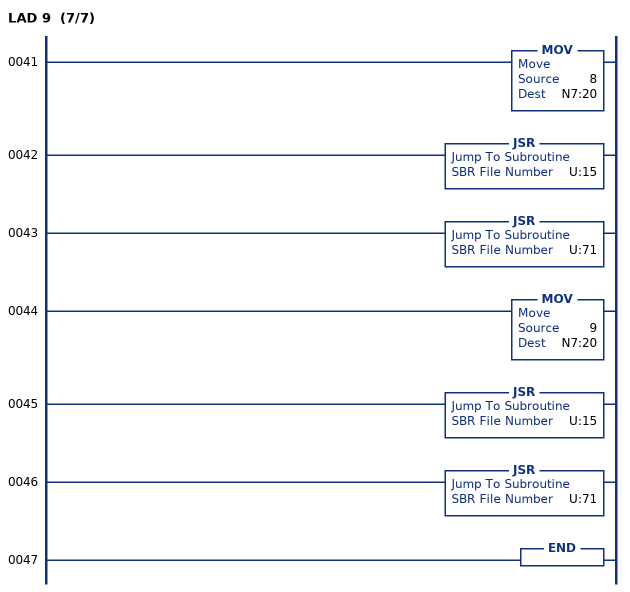
% Rung: 41 %
SOR MOV 8 N7:20 EOR
% Rung: 42 %
SOR JSR U:15 EOR
% Rung: 43 %
SOR JSR U:71 EOR
% Rung: 44 %
SOR MOV 9 N7:20 EOR
% Rung: 45 %
SOR JSR U:15 EOR
% Rung: 46 %
SOR JSR U:71 EOR
% Rung: 47 %
SOR END EOR

LADDER 10
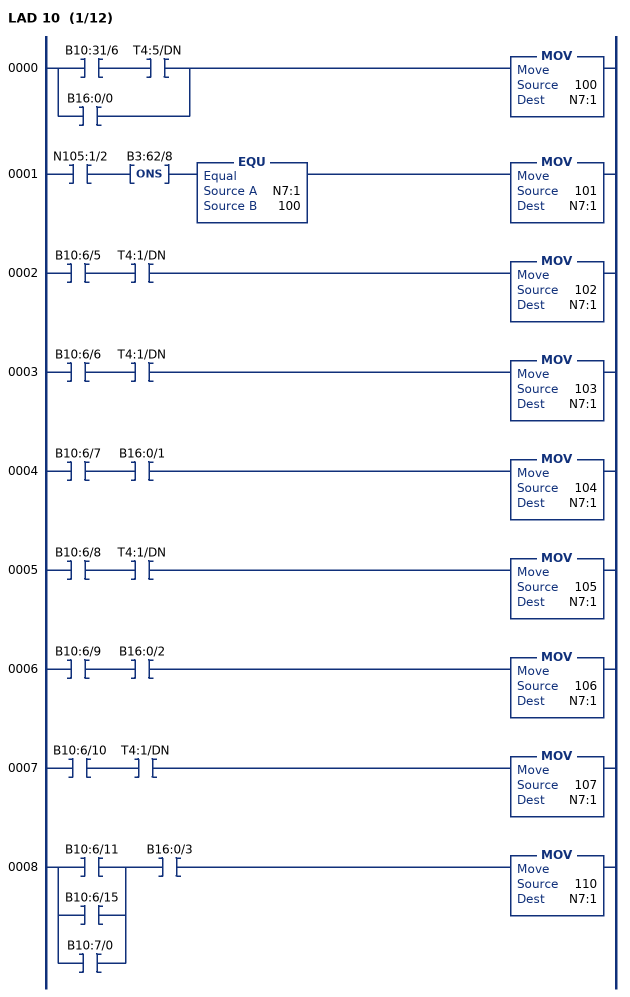
% Rung: 0 %
SOR BST XIC B10:31/6 XIC T4:5/DN NXB XIC B16:0/0 BND MOV 100 N7:1 EOR
% Rung: 1 %
SOR XIC N105:1/2 OSR B3:62/8 EQU N7:1 100 MOV 101 N7:1 EOR
% Rung: 2 %
SOR XIC B10:6/5 XIC T4:1/DN MOV 102 N7:1 EOR
% Rung: 3 %
SOR XIC B10:6/6 XIC T4:1/DN MOV 103 N7:1 EOR
% Rung: 4 %
SOR XIC B10:6/7 XIC B16:0/1 MOV 104 N7:1 EOR
% Rung: 5 %
SOR XIC B10:6/8 XIC T4:1/DN MOV 105 N7:1 EOR
% Rung: 6 %
SOR XIC B10:6/9 XIC B16:0/2 MOV 106 N7:1 EOR
% Rung: 7 %
SOR XIC B10:6/10 XIC T4:1/DN MOV 107 N7:1 EOR
% Rung: 8 %
SOR BST XIC B10:6/11 NXB XIC B10:6/15 NXB XIC B10:7/0 BND XIC B16:0/3 MOV 110 N7:1 EOR

